(* PLC project Unnamed, Unknown Unnamed 1 *)
(* stored: creationDateTime 2025-12-12T20:37:06, modificationDateTime 2025-12-12T21:30:29 *)

PROGRAM program2
  VAR
    Start AT %IX0.1 : BOOL;
    Stop AT %IX0.2 : BOOL;
    LED AT %QX0.1 : BOOL;
  END_VAR

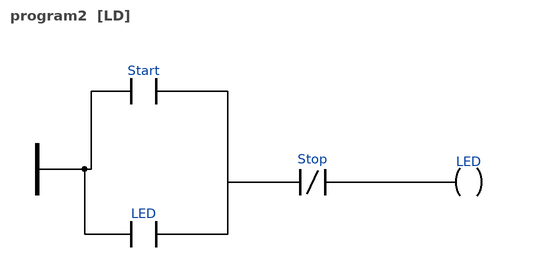
(* LD diagram, written out as Structured Text *)
LED := (LED OR Start) AND NOT Stop;
END_PROGRAM

CONFIGURATION Config0
  RESOURCE Res0 ON PLC
    TASK task0(INTERVAL := T#20ms, PRIORITY := 0);
    PROGRAM instance0 WITH task0 : program2;
  END_RESOURCE
END_CONFIGURATION
